INTERFACE I_AsynchronousRpcResponseFactory

METHOD PUBLIC TryCreate : BOOL
VAR_INPUT
	Destination : REFERENCE TO I_AsynchronousRpcResponse;
END_VAR
END_METHOD

END_INTERFACE

(* stored: Version 1.1.0.1, ProductVersion 3.1.4026.13
   Itf I_AsynchronousRpcResponseFactory: Id {3c6ebf61-433c-4639-9e6e-76c8248bd12a}
   Method TryCreate: Id {d1056d8d-b5c7-4c2c-a053-2fd3498ce0f5} *)
